{attribute 'GeneratedUsingTerminal: EK1100-0000-0018'}
{attribute addProperty BoxType "EK1100-0000-0018"}
{attribute addProperty Id "Beckhoff_EJ3xxxEK1122Beckhoff_EJ3xxxEK1122_1A5DA9A52A_0001_EJ3004_0000_0019EJ3004_CF76C88640A_0002_EJ3004_0000_0020EJ3004_CF76C88640A_0003_EJ3004_0000_0021EJ3004_CF76C88640A_0004_EJ3048_0000_0020EJ3048_FC58C0D676A_0005_EJ3058_0000_0020EJ3058_FC58C0D676A_0006_EJ3068_0000_0020EJ3068_FC58C0D676A_0007_EJ3068_0000_0021EJ3068_FC58C0D676A_0008_EJ3104_0000_0019EJ3104_BE8A5C9E44A_0009_EJ3104_0000_0020EJ3104_BE8A5C9E44A_0010_EJ3104_0000_0021EJ3104_BE8A5C9E44A_0011_EJ3108_0000_0017EJ3108_FC58C0D676A_0012_EJ3108_0000_0018EJ3108_84988DF084A_0013_EJ3108_0000_0019EJ3108_84988DF084A_0014_EJ3202_0000_0019EJ3202_353C76AA22A_0015_EJ3202_0000_0020EJ3202_353C76AA22A_0016_EJ3202_0000_0021EJ3202_353C76AA22A_0017_EJ3214_0000_0016EJ3214_65E7F5BB32A_0018_EJ3255_0000_0023EJ3255_0AE1D31454A_0019_EJ3318_0000_0017EJ3318_904F264374"}
{attribute addProperty CRC "2249408163"}
{attribute addProperty Size "1028"}
TYPE Beckhoff_EJ3xxx_86133EA3 EXTENDS EK1100_1FC0878B :
STRUCT
	{attribute addProperty Name "Beckhoff_EJ3xxxEK1122"}
	{attribute addProperty PreviousPort "Beckhoff EJ3xxx : B"}
	Beckhoff_EJ3xxxEK1122 : Beckhoff_EJ3xxxEK1122_1A5DA9A5;
	{attribute addProperty Name "A_0001_EJ3004_0000_0019"}
	{attribute addProperty PreviousPort "Beckhoff EJ3xxxEK1122 : C"}
	A_0001_EJ3004_0000_0019 : EJ3004_CF76C886;
	{attribute addProperty Name "A_0002_EJ3004_0000_0020"}
	{attribute addProperty PreviousPort "A_0001(EJ3004-0000-0019) : B"}
	A_0002_EJ3004_0000_0020 : EJ3004_CF76C886;
	{attribute addProperty Name "A_0003_EJ3004_0000_0021"}
	{attribute addProperty PreviousPort "A_0002(EJ3004-0000-0020) : B"}
	A_0003_EJ3004_0000_0021 : EJ3004_CF76C886;
	{attribute addProperty Name "A_0004_EJ3048_0000_0020"}
	{attribute addProperty PreviousPort "A_0003(EJ3004-0000-0021) : B"}
	A_0004_EJ3048_0000_0020 : EJ3048_FC58C0D6;
	{attribute addProperty Name "A_0005_EJ3058_0000_0020"}
	{attribute addProperty PreviousPort "A_0004(EJ3048-0000-0020) : B"}
	A_0005_EJ3058_0000_0020 : EJ3058_FC58C0D6;
	{attribute addProperty Name "A_0006_EJ3068_0000_0020"}
	{attribute addProperty PreviousPort "A_0005(EJ3058-0000-0020) : B"}
	A_0006_EJ3068_0000_0020 : EJ3068_FC58C0D6;
	{attribute addProperty Name "A_0007_EJ3068_0000_0021"}
	{attribute addProperty PreviousPort "A_0006(EJ3068-0000-0020) : B"}
	A_0007_EJ3068_0000_0021 : EJ3068_FC58C0D6;
	{attribute addProperty Name "A_0008_EJ3104_0000_0019"}
	{attribute addProperty PreviousPort "A_0007(EJ3068-0000-0021) : B"}
	A_0008_EJ3104_0000_0019 : EJ3104_BE8A5C9E;
	{attribute addProperty Name "A_0009_EJ3104_0000_0020"}
	{attribute addProperty PreviousPort "A_0008(EJ3104-0000-0019) : B"}
	A_0009_EJ3104_0000_0020 : EJ3104_BE8A5C9E;
	{attribute addProperty Name "A_0010_EJ3104_0000_0021"}
	{attribute addProperty PreviousPort "A_0009(EJ3104-0000-0020) : B"}
	A_0010_EJ3104_0000_0021 : EJ3104_BE8A5C9E;
	{attribute addProperty Name "A_0011_EJ3108_0000_0017"}
	{attribute addProperty PreviousPort "A_0010(EJ3104-0000-0021) : B"}
	A_0011_EJ3108_0000_0017 : EJ3108_FC58C0D6;
	{attribute addProperty Name "A_0012_EJ3108_0000_0018"}
	{attribute addProperty PreviousPort "A_0011(EJ3108-0000-0017) : B"}
	A_0012_EJ3108_0000_0018 : EJ3108_84988DF0;
	{attribute addProperty Name "A_0013_EJ3108_0000_0019"}
	{attribute addProperty PreviousPort "A_0012(EJ3108-0000-0018) : B"}
	A_0013_EJ3108_0000_0019 : EJ3108_84988DF0;
	{attribute addProperty Name "A_0014_EJ3202_0000_0019"}
	{attribute addProperty PreviousPort "A_0013(EJ3108-0000-0019) : B"}
	A_0014_EJ3202_0000_0019 : EJ3202_353C76AA;
	{attribute addProperty Name "A_0015_EJ3202_0000_0020"}
	{attribute addProperty PreviousPort "A_0014(EJ3202-0000-0019) : B"}
	A_0015_EJ3202_0000_0020 : EJ3202_353C76AA;
	{attribute addProperty Name "A_0016_EJ3202_0000_0021"}
	{attribute addProperty PreviousPort "A_0015(EJ3202-0000-0020) : B"}
	A_0016_EJ3202_0000_0021 : EJ3202_353C76AA;
	{attribute addProperty Name "A_0017_EJ3214_0000_0016"}
	{attribute addProperty PreviousPort "A_0016(EJ3202-0000-0021) : B"}
	A_0017_EJ3214_0000_0016 : EJ3214_65E7F5BB;
	{attribute addProperty Name "A_0018_EJ3255_0000_0023"}
	{attribute addProperty PreviousPort "A_0017(EJ3214-0000-0016) : B"}
	A_0018_EJ3255_0000_0023 : EJ3255_0AE1D314;
	{attribute addProperty Name "A_0019_EJ3318_0000_0017"}
	{attribute addProperty PreviousPort "A_0018(EJ3255-0000-0023) : B"}
	A_0019_EJ3318_0000_0017 : EJ3318_904F2643;
END_STRUCT
END_TYPE

(* stored: Version 1.2.0.0, ProductVersion 3.1.4024.9
   DUT Beckhoff_EJ3xxx_86133EA3: Id {2c4af25d-89e9-4c44-a395-72b5884f5ad1} *)
